FUNCTION F_Round_REAL : REAL
VAR_INPUT
	rInReal			: REAL;
	iPrecision		: INT;
END_VAR
VAR
	rOutReal		: REAL;
	rRoundingVal	: REAL; //last digit for rounding purposes
END_VAR

IF RealIsNaN(rInReal) THEN
	RETURN;
END_IF

rOutReal := rInReal * EXPT(10,ABS(iPrecision));

rRoundingVal := rOutReal - DINT_TO_REAL(TRUNC(rOutReal));
IF rRoundingVal >= 0.5 THEN
	rOutReal	:= DINT_TO_REAL(TRUNC(rOutReal)) + 1;
ELSIF rRoundingVal <= -0.5 THEN
	rOutReal	:= DINT_TO_REAL(TRUNC(rOutReal)) - 1;
ELSE
	rOutReal	:= DINT_TO_REAL(TRUNC(rOutReal));
END_IF

F_Round_REAL	:= rOutReal / EXPT(10,ABS(iPrecision));

END_FUNCTION

(* stored: Version 1.1.0.1, ProductVersion 3.1.4024.12
   POU F_Round_REAL: Id {b9cf1da4-c3b2-46c2-bd68-9a65f318233e}, SpecialFunc None *)
